INTERFACE PUBLIC I_AsyncCommand extends I_Command

METHOD PUBLIC Abort
END_METHOD

METHOD PUBLIC CyclicCall
END_METHOD

{attribute 'monitoring' := 'call'}
PROPERTY PUBLIC Executing : BOOL
GET
END_GET
END_PROPERTY

METHOD PUBLIC GetResult : I_Result
END_METHOD

{attribute 'monitoring' := 'call'}
PROPERTY PUBLIC Idle : BOOL
GET
END_GET
END_PROPERTY

{attribute 'monitoring' := 'call'}
PROPERTY PUBLIC Stopped : BOOL
GET
END_GET
END_PROPERTY

END_INTERFACE

(* stored: Version 1.1.0.1, ProductVersion 3.1.4024.12
   Itf I_AsyncCommand: Id {1bee37c0-c3a5-0b6f-13cb-01d3f3ae4d04}
   Method Abort: Id {af0faec8-03c9-094f-32c6-8876a661ccc2}
   Method CyclicCall: Id {33296f58-4355-0dfc-3db1-1173b9e296e6}
   Property Executing: Id {80e6bff9-9cee-4b2e-8046-11c9af1f56f5}
   Get Get: Id {e5f7b0fa-03c1-4f63-b93a-6244a2deed6b}
   Method GetResult: Id {7e02e640-00d8-4d83-bbea-a01774cf5b32}
   Property Idle: Id {d35c522f-d4b4-4764-9245-33fcfc9af43d}
   Get Get: Id {3cdd3b59-67b1-4cfd-97d1-15caf9b65b77}
   Property Stopped: Id {6becda4a-e9b2-4c88-ae7c-dd90703c5712}
   Get Get: Id {217bf73d-8f76-4ae0-bf6e-7c029310b2a8} *)
